(* PLC project KinIn_v3.project, CODESYS CODESYS V3.5 SP19 *)
(* stored: creationDateTime 2025-01-20T16:27:17.0506241, modificationDateTime 2025-01-20T16:17:39.6822999 *)

FUNCTION_BLOCK isValueNegligible
  VAR_INPUT
    {attribute 'variable_length_array_original_scope' := 'Inout'}
    {attribute 'variable_length_array' := 'ARRAY[*] OF REAL'}
    {attribute 'Dimensions' := '1'}
    nearArray : POINTER TO REAL;  (* scalar *)
  END_VAR
  VAR_OUTPUT
    judge : INT;
  END_VAR
  VAR
    norm : norm;
    normVal : REAL;
  END_VAR

            norm(vector:= nearArray, normValue=> normVal);
IF normVal< 0.0000001 THEN
	judge:=1;
ELSE
	judge:=0;
END_IF

          
END_FUNCTION_BLOCK
